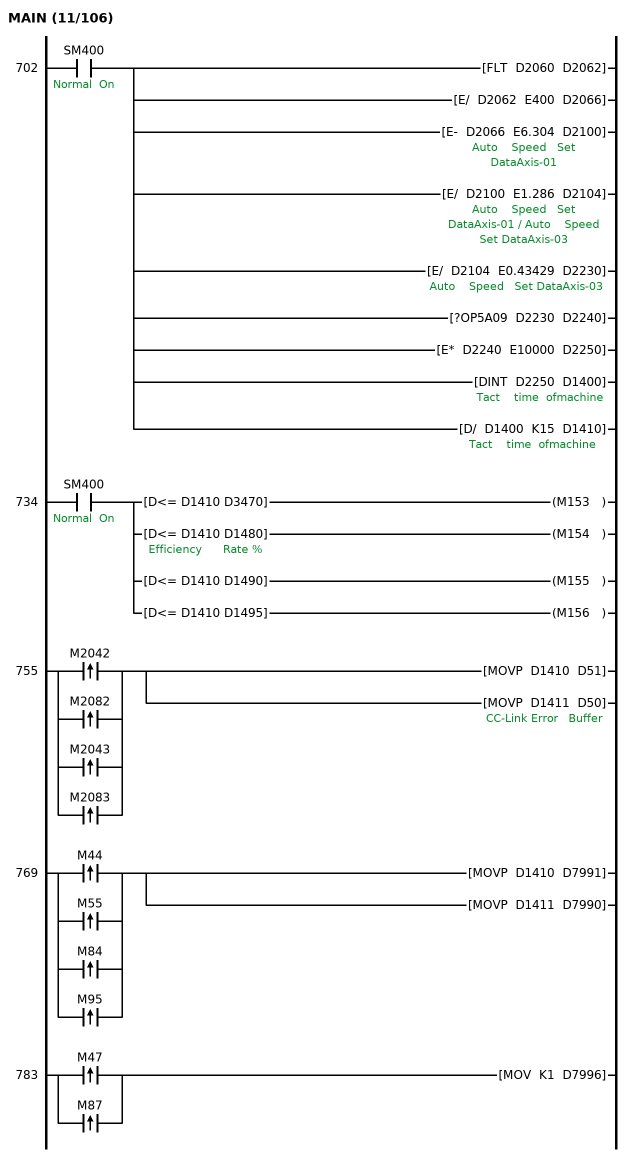
[picture p288: ladder of MAIN, rungs at steps 702 to 783]
702   LD      SM400  ; Normal  On
      FLT     D2060 D2062
      E/      D2062 E400 D2066
      E-      D2066 E6.304 D2100  ; Auto    Speed   Set DataAxis-01
      E/      D2100 E1.286 D2104  ; Auto    Speed   Set DataAxis-03
      E/      D2104 E0.43429 D2230
      ?OP5A09 D2230 D2240
      E*      D2240 E10000 D2250
      DINT    D2250 D1400  ; Tact    time  ofmachine
      D/      D1400 K15 D1410
734   LD      SM400  ; Normal  On
      MPS
      ANDD<=  D1410 D3470
      OUT     M153
      MRD
      ANDD<=  D1410 D1480  ; Efficiency      Rate %
      OUT     M154
      MRD
      ANDD<=  D1410 D1490
      OUT     M155
      MPP
      ANDD<=  D1410 D1495
      OUT     M156
755   LDP     M2042
      ORP     M2082
      ORP     M2043
      ORP     M2083
      MOVP    D1410 D51
      MOVP    D1411 D50  ; CC-Link Error   Buffer
769   LDP     M44
      ORP     M55
      ORP     M84
      ORP     M95
      MOVP    D1410 D7991
      MOVP    D1411 D7990
783   LDP     M47
      ORP     M87
      MOV     K1 D7996
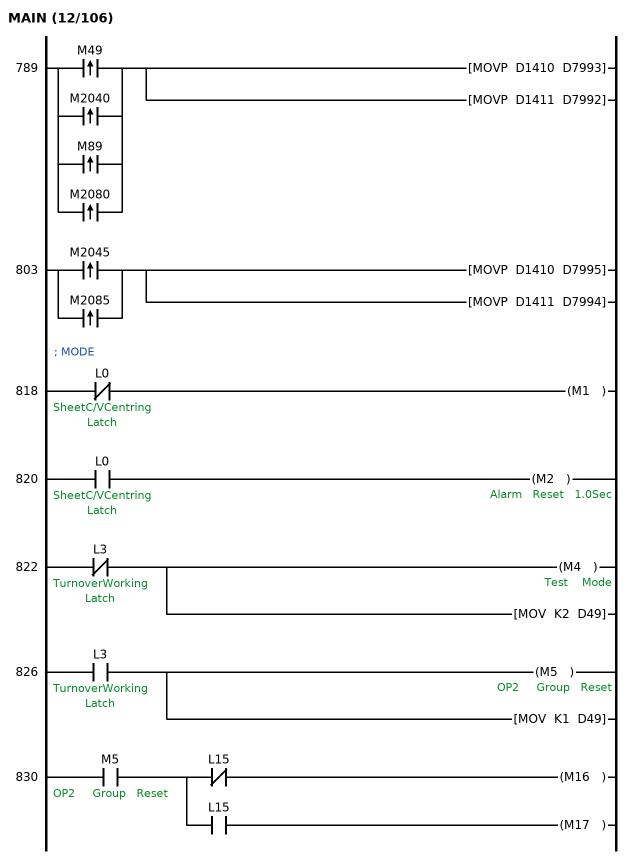
789   LDP     M49
      ORP     M2040
      ORP     M89
      ORP     M2080
      MOVP    D1410 D7993
      MOVP    D1411 D7992
803   LDP     M2045
      ORP     M2085
      MOVP    D1410 D7995
      MOVP    D1411 D7994
; MODE
818   LDI     L0  ; SheetC/VCentringLatch
      OUT     M1
820   LD      L0  ; SheetC/VCentringLatch
      OUT     M2  ; Alarm   Reset   1.0Sec
822   LDI     L3  ; TurnoverWorking Latch
      OUT     M4  ; Test    Mode
      MOV     K2 D49
826   LD      L3  ; TurnoverWorking Latch
      OUT     M5  ; OP2     Group   Reset
      MOV     K1 D49
830   LD      M5  ; OP2     Group   Reset
      MPS
      ANI     L15
      OUT     M16
      MPP
      AND     L15
      OUT     M17
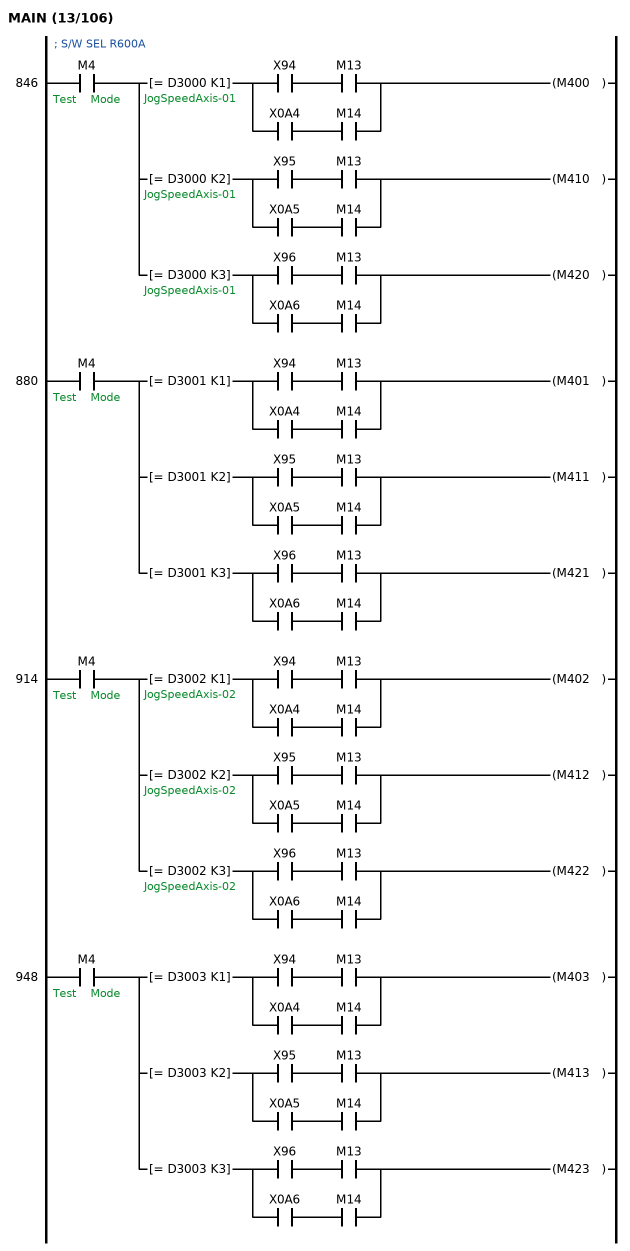
; S/W SEL R600A
846   LD      M4  ; Test    Mode
      MPS
      AND=    D3000 K1  ; JogSpeedAxis-01
      LD      X94
      AND     M13
      LD      X0A4
      AND     M14
      ORB
      ANB
      OUT     M400
      MRD
      AND=    D3000 K2  ; JogSpeedAxis-01
      LD      X95
      AND     M13
      LD      X0A5
      AND     M14
      ORB
      ANB
      OUT     M410
      MPP
      AND=    D3000 K3  ; JogSpeedAxis-01
      LD      X96
      AND     M13
      LD      X0A6
      AND     M14
      ORB
      ANB
      OUT     M420
880   LD      M4  ; Test    Mode
      MPS
      AND=    D3001 K1
      LD      X94
      AND     M13
      LD      X0A4
      AND     M14
      ORB
      ANB
      OUT     M401
      MRD
      AND=    D3001 K2
      LD      X95
      AND     M13
      LD      X0A5
      AND     M14
      ORB
      ANB
      OUT     M411
      MPP
      AND=    D3001 K3
      LD      X96
      AND     M13
      LD      X0A6
      AND     M14
      ORB
      ANB
      OUT     M421
914   LD      M4  ; Test    Mode
      MPS
      AND=    D3002 K1  ; JogSpeedAxis-02
      LD      X94
      AND     M13
      LD      X0A4
      AND     M14
      ORB
      ANB
      OUT     M402
      MRD
      AND=    D3002 K2  ; JogSpeedAxis-02
      LD      X95
      AND     M13
      LD      X0A5
      AND     M14
      ORB
      ANB
      OUT     M412
      MPP
      AND=    D3002 K3  ; JogSpeedAxis-02
      LD      X96
      AND     M13
      LD      X0A6
      AND     M14
      ORB
      ANB
      OUT     M422
948   LD      M4  ; Test    Mode
      MPS
      AND=    D3003 K1
      LD      X94
      AND     M13
      LD      X0A4
      AND     M14
      ORB
      ANB
      OUT     M403
      MRD
      AND=    D3003 K2
      LD      X95
      AND     M13
      LD      X0A5
      AND     M14
      ORB
      ANB
      OUT     M413
      MPP
      AND=    D3003 K3
      LD      X96
      AND     M13
      LD      X0A6
      AND     M14
      ORB
      ANB
      OUT     M423
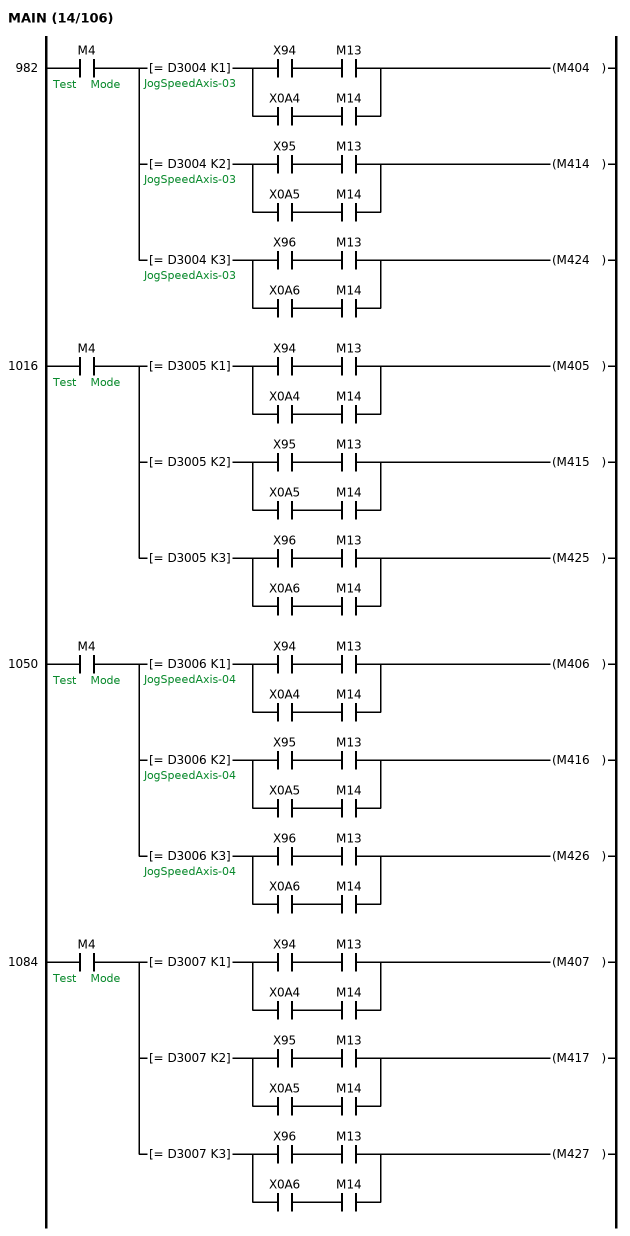
982   LD      M4  ; Test    Mode
      MPS
      AND=    D3004 K1  ; JogSpeedAxis-03
      LD      X94
      AND     M13
      LD      X0A4
      AND     M14
      ORB
      ANB
      OUT     M404
      MRD
      AND=    D3004 K2  ; JogSpeedAxis-03
      LD      X95
      AND     M13
      LD      X0A5
      AND     M14
      ORB
      ANB
      OUT     M414
      MPP
      AND=    D3004 K3  ; JogSpeedAxis-03
      LD      X96
      AND     M13
      LD      X0A6
      AND     M14
      ORB
      ANB
      OUT     M424
1016  LD      M4  ; Test    Mode
      MPS
      AND=    D3005 K1
      LD      X94
      AND     M13
      LD      X0A4
      AND     M14
      ORB
      ANB
      OUT     M405
      MRD
      AND=    D3005 K2
      LD      X95
      AND     M13
      LD      X0A5
      AND     M14
      ORB
      ANB
      OUT     M415
      MPP
      AND=    D3005 K3
      LD      X96
      AND     M13
      LD      X0A6
      AND     M14
      ORB
      ANB
      OUT     M425
1050  LD      M4  ; Test    Mode
      MPS
      AND=    D3006 K1  ; JogSpeedAxis-04
      LD      X94
      AND     M13
      LD      X0A4
      AND     M14
      ORB
      ANB
      OUT     M406
      MRD
      AND=    D3006 K2  ; JogSpeedAxis-04
      LD      X95
      AND     M13
      LD      X0A5
      AND     M14
      ORB
      ANB
      OUT     M416
      MPP
      AND=    D3006 K3  ; JogSpeedAxis-04
      LD      X96
      AND     M13
      LD      X0A6
      AND     M14
      ORB
      ANB
      OUT     M426
1084  LD      M4  ; Test    Mode
      MPS
      AND=    D3007 K1
      LD      X94
      AND     M13
      LD      X0A4
      AND     M14
      ORB
      ANB
      OUT     M407
      MRD
      AND=    D3007 K2
      LD      X95
      AND     M13
      LD      X0A5
      AND     M14
      ORB
      ANB
      OUT     M417
      MPP
      AND=    D3007 K3
      LD      X96
      AND     M13
      LD      X0A6
      AND     M14
      ORB
      ANB
      OUT     M427
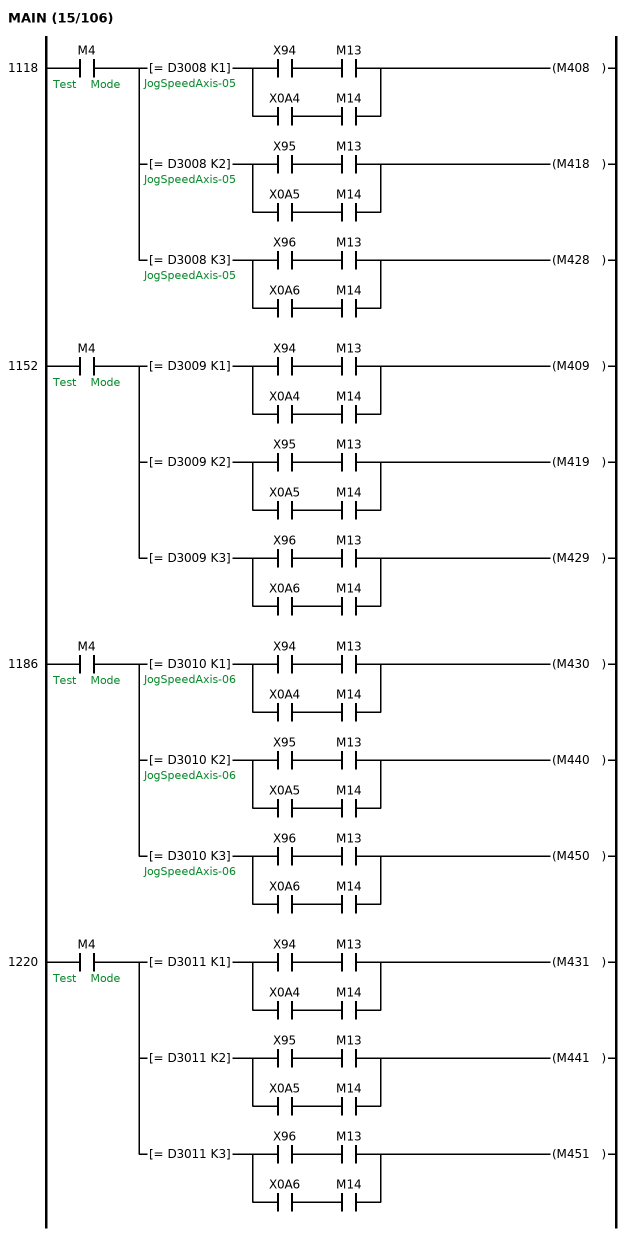
1118  LD      M4  ; Test    Mode
      MPS
      AND=    D3008 K1  ; JogSpeedAxis-05
      LD      X94
      AND     M13
      LD      X0A4
      AND     M14
      ORB
      ANB
      OUT     M408
      MRD
      AND=    D3008 K2  ; JogSpeedAxis-05
      LD      X95
      AND     M13
      LD      X0A5
      AND     M14
      ORB
      ANB
      OUT     M418
      MPP
      AND=    D3008 K3  ; JogSpeedAxis-05
      LD      X96
      AND     M13
      LD      X0A6
      AND     M14
      ORB
      ANB
      OUT     M428
1152  LD      M4  ; Test    Mode
      MPS
      AND=    D3009 K1
      LD      X94
      AND     M13
      LD      X0A4
      AND     M14
      ORB
      ANB
      OUT     M409
      MRD
      AND=    D3009 K2
      LD      X95
      AND     M13
      LD      X0A5
      AND     M14
      ORB
      ANB
      OUT     M419
      MPP
      AND=    D3009 K3
      LD      X96
      AND     M13
      LD      X0A6
      AND     M14
      ORB
      ANB
      OUT     M429
1186  LD      M4  ; Test    Mode
      MPS
      AND=    D3010 K1  ; JogSpeedAxis-06
      LD      X94
      AND     M13
      LD      X0A4
      AND     M14
      ORB
      ANB
      OUT     M430
      MRD
      AND=    D3010 K2  ; JogSpeedAxis-06
      LD      X95
      AND     M13
      LD      X0A5
      AND     M14
      ORB
      ANB
      OUT     M440
      MPP
      AND=    D3010 K3  ; JogSpeedAxis-06
      LD      X96
      AND     M13
      LD      X0A6
      AND     M14
      ORB
      ANB
      OUT     M450
1220  LD      M4  ; Test    Mode
      MPS
      AND=    D3011 K1
      LD      X94
      AND     M13
      LD      X0A4
      AND     M14
      ORB
      ANB
      OUT     M431
      MRD
      AND=    D3011 K2
      LD      X95
      AND     M13
      LD      X0A5
      AND     M14
      ORB
      ANB
      OUT     M441
      MPP
      AND=    D3011 K3
      LD      X96
      AND     M13
      LD      X0A6
      AND     M14
      ORB
      ANB
      OUT     M451
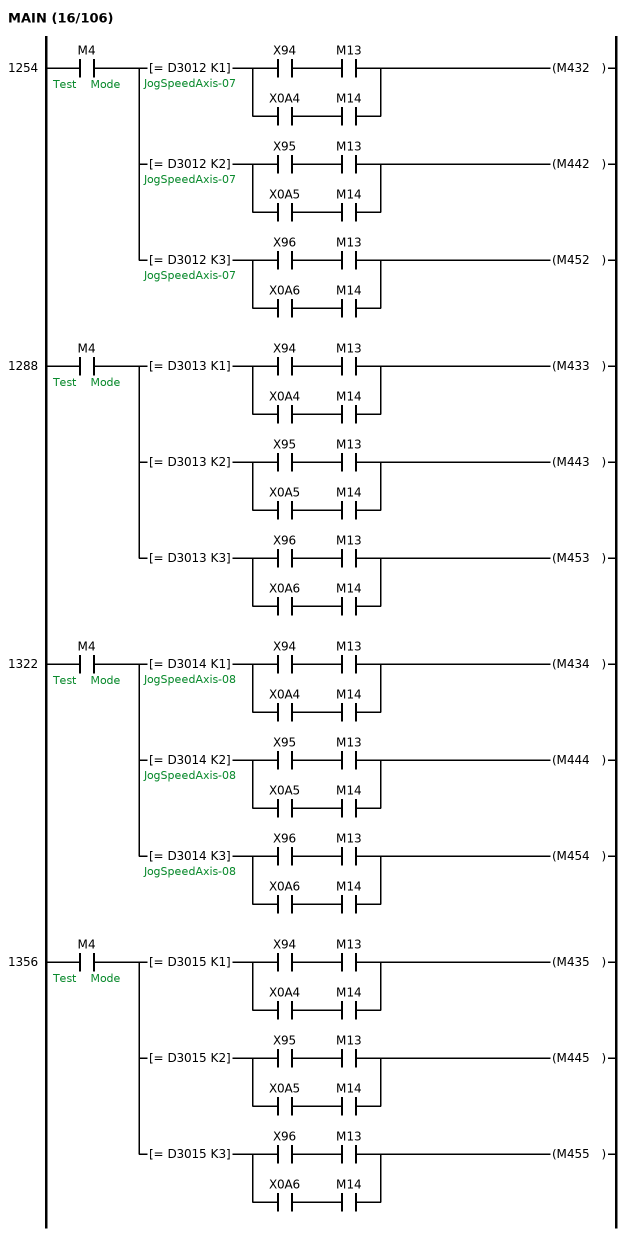
1254  LD      M4  ; Test    Mode
      MPS
      AND=    D3012 K1  ; JogSpeedAxis-07
      LD      X94
      AND     M13
      LD      X0A4
      AND     M14
      ORB
      ANB
      OUT     M432
      MRD
      AND=    D3012 K2  ; JogSpeedAxis-07
      LD      X95
      AND     M13
      LD      X0A5
      AND     M14
      ORB
      ANB
      OUT     M442
      MPP
      AND=    D3012 K3  ; JogSpeedAxis-07
      LD      X96
      AND     M13
      LD      X0A6
      AND     M14
      ORB
      ANB
      OUT     M452
1288  LD      M4  ; Test    Mode
      MPS
      AND=    D3013 K1
      LD      X94
      AND     M13
      LD      X0A4
      AND     M14
      ORB
      ANB
      OUT     M433
      MRD
      AND=    D3013 K2
      LD      X95
      AND     M13
      LD      X0A5
      AND     M14
      ORB
      ANB
      OUT     M443
      MPP
      AND=    D3013 K3
      LD      X96
      AND     M13
      LD      X0A6
      AND     M14
      ORB
      ANB
      OUT     M453
1322  LD      M4  ; Test    Mode
      MPS
      AND=    D3014 K1  ; JogSpeedAxis-08
      LD      X94
      AND     M13
      LD      X0A4
      AND     M14
      ORB
      ANB
      OUT     M434
      MRD
      AND=    D3014 K2  ; JogSpeedAxis-08
      LD      X95
      AND     M13
      LD      X0A5
      AND     M14
      ORB
      ANB
      OUT     M444
      MPP
      AND=    D3014 K3  ; JogSpeedAxis-08
      LD      X96
      AND     M13
      LD      X0A6
      AND     M14
      ORB
      ANB
      OUT     M454
1356  LD      M4  ; Test    Mode
      MPS
      AND=    D3015 K1
      LD      X94
      AND     M13
      LD      X0A4
      AND     M14
      ORB
      ANB
      OUT     M435
      MRD
      AND=    D3015 K2
      LD      X95
      AND     M13
      LD      X0A5
      AND     M14
      ORB
      ANB
      OUT     M445
      MPP
      AND=    D3015 K3
      LD      X96
      AND     M13
      LD      X0A6
      AND     M14
      ORB
      ANB
      OUT     M455
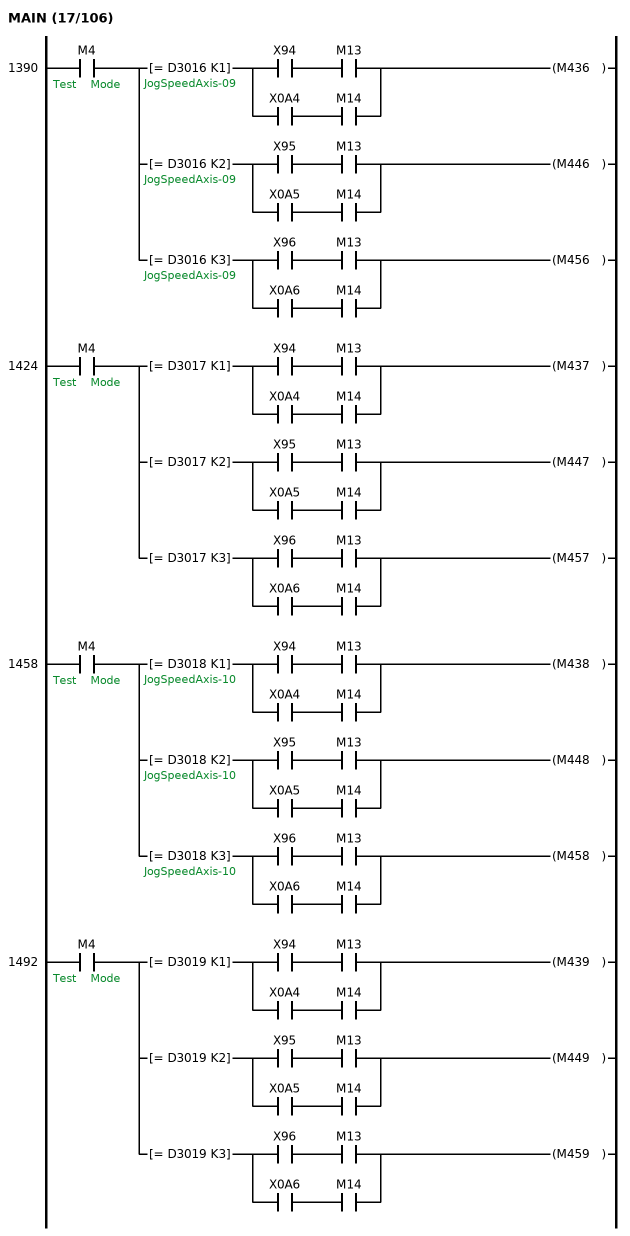
1390  LD      M4  ; Test    Mode
      MPS
      AND=    D3016 K1  ; JogSpeedAxis-09
      LD      X94
      AND     M13
      LD      X0A4
      AND     M14
      ORB
      ANB
      OUT     M436
      MRD
      AND=    D3016 K2  ; JogSpeedAxis-09
      LD      X95
      AND     M13
      LD      X0A5
      AND     M14
      ORB
      ANB
      OUT     M446
      MPP
      AND=    D3016 K3  ; JogSpeedAxis-09
      LD      X96
      AND     M13
      LD      X0A6
      AND     M14
      ORB
      ANB
      OUT     M456
1424  LD      M4  ; Test    Mode
      MPS
      AND=    D3017 K1
      LD      X94
      AND     M13
      LD      X0A4
      AND     M14
      ORB
      ANB
      OUT     M437
      MRD
      AND=    D3017 K2
      LD      X95
      AND     M13
      LD      X0A5
      AND     M14
      ORB
      ANB
      OUT     M447
      MPP
      AND=    D3017 K3
      LD      X96
      AND     M13
      LD      X0A6
      AND     M14
      ORB
      ANB
      OUT     M457
1458  LD      M4  ; Test    Mode
      MPS
      AND=    D3018 K1  ; JogSpeedAxis-10
      LD      X94
      AND     M13
      LD      X0A4
      AND     M14
      ORB
      ANB
      OUT     M438
      MRD
      AND=    D3018 K2  ; JogSpeedAxis-10
      LD      X95
      AND     M13
      LD      X0A5
      AND     M14
      ORB
      ANB
      OUT     M448
      MPP
      AND=    D3018 K3  ; JogSpeedAxis-10
      LD      X96
      AND     M13
      LD      X0A6
      AND     M14
      ORB
      ANB
      OUT     M458
1492  LD      M4  ; Test    Mode
      MPS
      AND=    D3019 K1
      LD      X94
      AND     M13
      LD      X0A4
      AND     M14
      ORB
      ANB
      OUT     M439
      MRD
      AND=    D3019 K2
      LD      X95
      AND     M13
      LD      X0A5
      AND     M14
      ORB
      ANB
      OUT     M449
      MPP
      AND=    D3019 K3
      LD      X96
      AND     M13
      LD      X0A6
      AND     M14
      ORB
      ANB
      OUT     M459
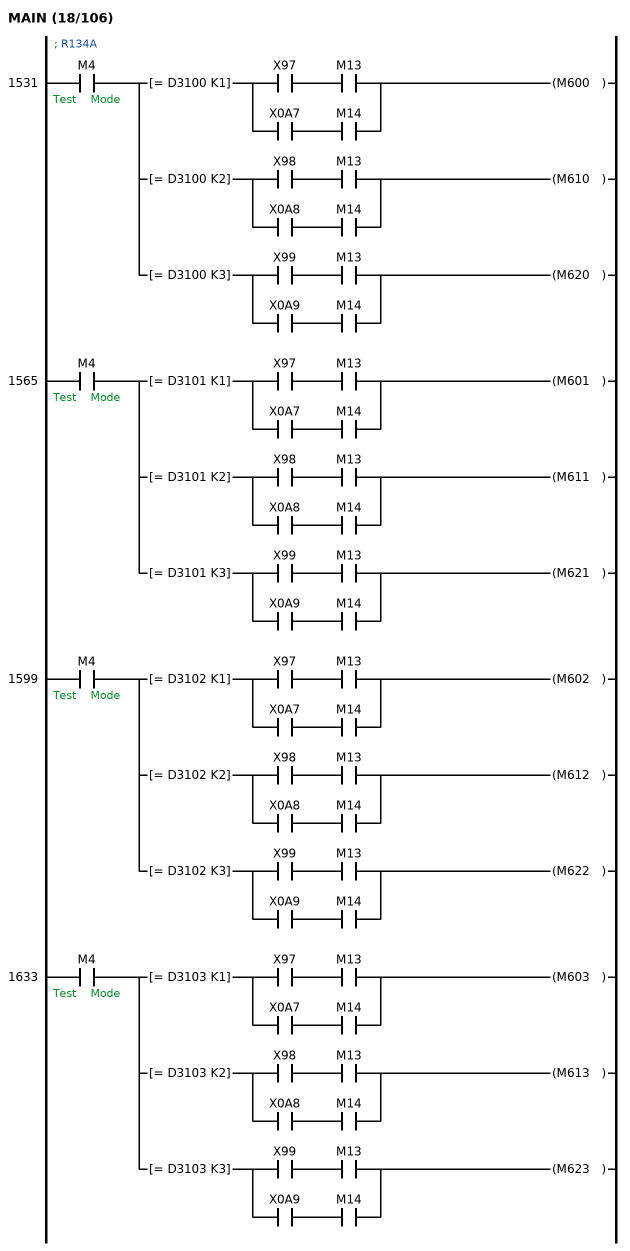
; R134A
1531  LD      M4  ; Test    Mode
      MPS
      AND=    D3100 K1
      LD      X97
      AND     M13
      LD      X0A7
      AND     M14
      ORB
      ANB
      OUT     M600
      MRD
      AND=    D3100 K2
      LD      X98
      AND     M13
      LD      X0A8
      AND     M14
      ORB
      ANB
      OUT     M610
      MPP
      AND=    D3100 K3
      LD      X99
      AND     M13
      LD      X0A9
      AND     M14
      ORB
      ANB
      OUT     M620
1565  LD      M4  ; Test    Mode
      MPS
      AND=    D3101 K1
      LD      X97
      AND     M13
      LD      X0A7
      AND     M14
      ORB
      ANB
      OUT     M601
      MRD
      AND=    D3101 K2
      LD      X98
      AND     M13
      LD      X0A8
      AND     M14
      ORB
      ANB
      OUT     M611
      MPP
      AND=    D3101 K3
      LD      X99
      AND     M13
      LD      X0A9
      AND     M14
      ORB
      ANB
      OUT     M621
1599  LD      M4  ; Test    Mode
      MPS
      AND=    D3102 K1
      LD      X97
      AND     M13
      LD      X0A7
      AND     M14
      ORB
      ANB
      OUT     M602
      MRD
      AND=    D3102 K2
      LD      X98
      AND     M13
      LD      X0A8
      AND     M14
      ORB
      ANB
      OUT     M612
      MPP
      AND=    D3102 K3
      LD      X99
      AND     M13
      LD      X0A9
      AND     M14
      ORB
      ANB
      OUT     M622
1633  LD      M4  ; Test    Mode
      MPS
      AND=    D3103 K1
      LD      X97
      AND     M13
      LD      X0A7
      AND     M14
      ORB
      ANB
      OUT     M603
      MRD
      AND=    D3103 K2
      LD      X98
      AND     M13
      LD      X0A8
      AND     M14
      ORB
      ANB
      OUT     M613
      MPP
      AND=    D3103 K3
      LD      X99
      AND     M13
      LD      X0A9
      AND     M14
      ORB
      ANB
      OUT     M623
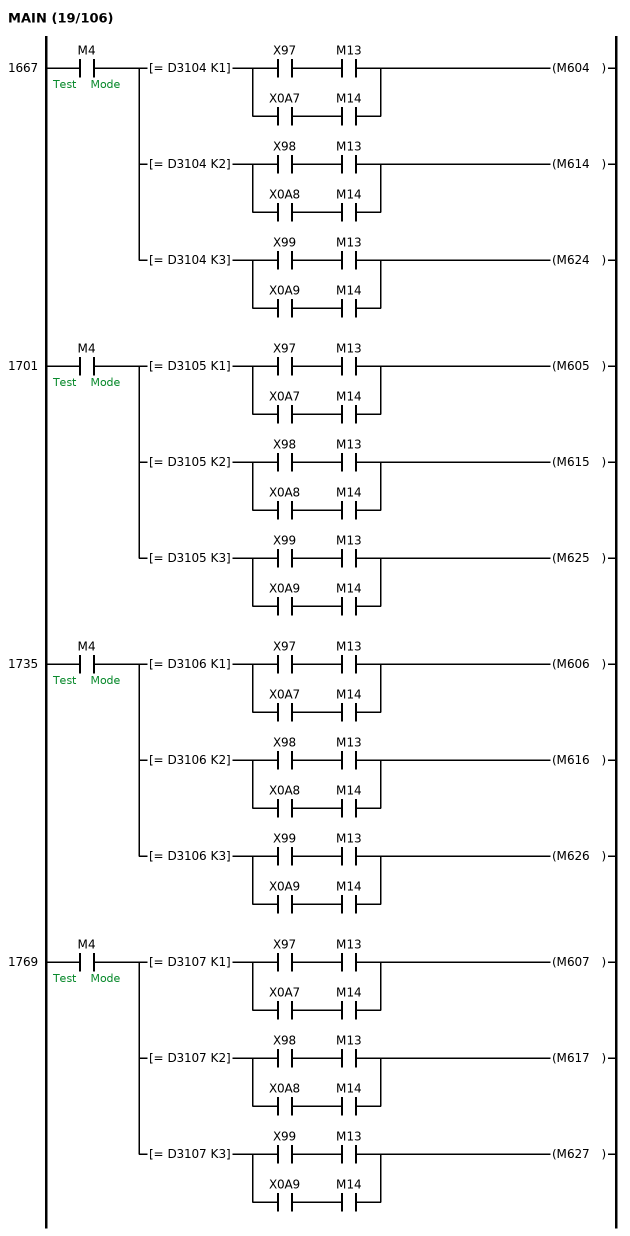
1667  LD      M4  ; Test    Mode
      MPS
      AND=    D3104 K1
      LD      X97
      AND     M13
      LD      X0A7
      AND     M14
      ORB
      ANB
      OUT     M604
      MRD
      AND=    D3104 K2
      LD      X98
      AND     M13
      LD      X0A8
      AND     M14
      ORB
      ANB
      OUT     M614
      MPP
      AND=    D3104 K3
      LD      X99
      AND     M13
      LD      X0A9
      AND     M14
      ORB
      ANB
      OUT     M624
1701  LD      M4  ; Test    Mode
      MPS
      AND=    D3105 K1
      LD      X97
      AND     M13
      LD      X0A7
      AND     M14
      ORB
      ANB
      OUT     M605
      MRD
      AND=    D3105 K2
      LD      X98
      AND     M13
      LD      X0A8
      AND     M14
      ORB
      ANB
      OUT     M615
      MPP
      AND=    D3105 K3
      LD      X99
      AND     M13
      LD      X0A9
      AND     M14
      ORB
      ANB
      OUT     M625
1735  LD      M4  ; Test    Mode
      MPS
      AND=    D3106 K1
      LD      X97
      AND     M13
      LD      X0A7
      AND     M14
      ORB
      ANB
      OUT     M606
      MRD
      AND=    D3106 K2
      LD      X98
      AND     M13
      LD      X0A8
      AND     M14
      ORB
      ANB
      OUT     M616
      MPP
      AND=    D3106 K3
      LD      X99
      AND     M13
      LD      X0A9
      AND     M14
      ORB
      ANB
      OUT     M626
1769  LD      M4  ; Test    Mode
      MPS
      AND=    D3107 K1
      LD      X97
      AND     M13
      LD      X0A7
      AND     M14
      ORB
      ANB
      OUT     M607
      MRD
      AND=    D3107 K2
      LD      X98
      AND     M13
      LD      X0A8
      AND     M14
      ORB
      ANB
      OUT     M617
      MPP
      AND=    D3107 K3
      LD      X99
      AND     M13
      LD      X0A9
      AND     M14
      ORB
      ANB
      OUT     M627
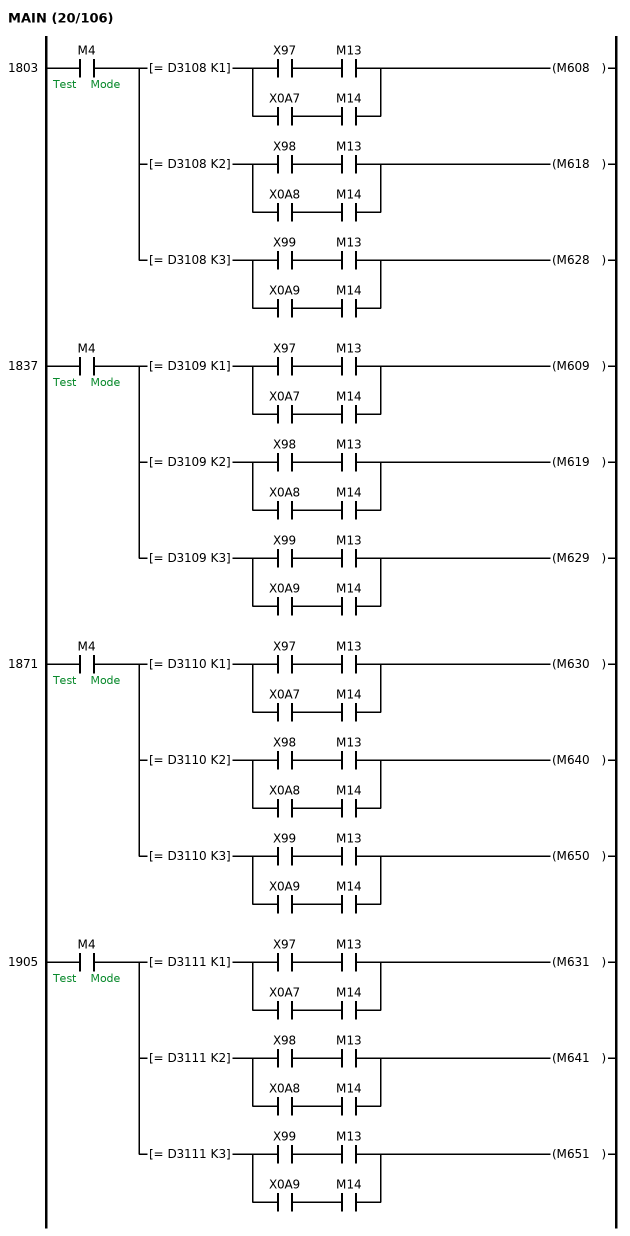
1803  LD      M4  ; Test    Mode
      MPS
      AND=    D3108 K1
      LD      X97
      AND     M13
      LD      X0A7
      AND     M14
      ORB
      ANB
      OUT     M608
      MRD
      AND=    D3108 K2
      LD      X98
      AND     M13
      LD      X0A8
      AND     M14
      ORB
      ANB
      OUT     M618
      MPP
      AND=    D3108 K3
      LD      X99
      AND     M13
      LD      X0A9
      AND     M14
      ORB
      ANB
      OUT     M628
1837  LD      M4  ; Test    Mode
      MPS
      AND=    D3109 K1
      LD      X97
      AND     M13
      LD      X0A7
      AND     M14
      ORB
      ANB
      OUT     M609
      MRD
      AND=    D3109 K2
      LD      X98
      AND     M13
      LD      X0A8
      AND     M14
      ORB
      ANB
      OUT     M619
      MPP
      AND=    D3109 K3
      LD      X99
      AND     M13
      LD      X0A9
      AND     M14
      ORB
      ANB
      OUT     M629
1871  LD      M4  ; Test    Mode
      MPS
      AND=    D3110 K1
      LD      X97
      AND     M13
      LD      X0A7
      AND     M14
      ORB
      ANB
      OUT     M630
      MRD
      AND=    D3110 K2
      LD      X98
      AND     M13
      LD      X0A8
      AND     M14
      ORB
      ANB
      OUT     M640
      MPP
      AND=    D3110 K3
      LD      X99
      AND     M13
      LD      X0A9
      AND     M14
      ORB
      ANB
      OUT     M650
1905  LD      M4  ; Test    Mode
      MPS
      AND=    D3111 K1
      LD      X97
      AND     M13
      LD      X0A7
      AND     M14
      ORB
      ANB
      OUT     M631
      MRD
      AND=    D3111 K2
      LD      X98
      AND     M13
      LD      X0A8
      AND     M14
      ORB
      ANB
      OUT     M641
      MPP
      AND=    D3111 K3
      LD      X99
      AND     M13
      LD      X0A9
      AND     M14
      ORB
      ANB
      OUT     M651
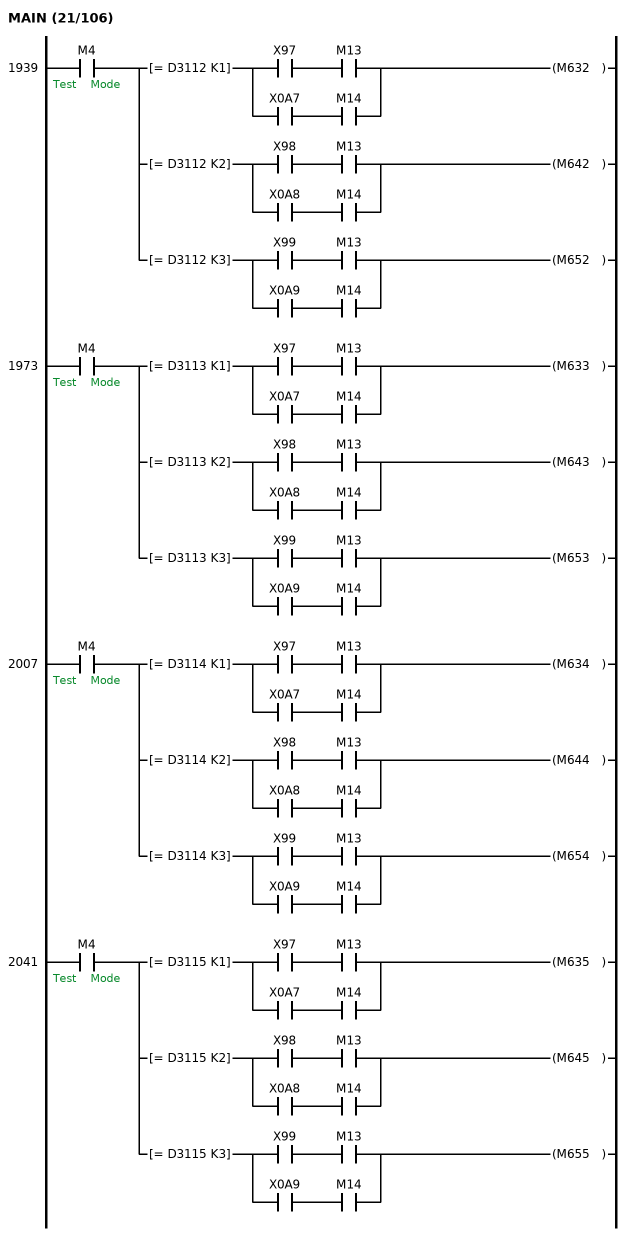
1939  LD      M4  ; Test    Mode
      MPS
      AND=    D3112 K1
      LD      X97
      AND     M13
      LD      X0A7
      AND     M14
      ORB
      ANB
      OUT     M632
      MRD
      AND=    D3112 K2
      LD      X98
      AND     M13
      LD      X0A8
      AND     M14
      ORB
      ANB
      OUT     M642
      MPP
      AND=    D3112 K3
      LD      X99
      AND     M13
      LD      X0A9
      AND     M14
      ORB
      ANB
      OUT     M652
1973  LD      M4  ; Test    Mode
      MPS
      AND=    D3113 K1
      LD      X97
      AND     M13
      LD      X0A7
      AND     M14
      ORB
      ANB
      OUT     M633
      MRD
      AND=    D3113 K2
      LD      X98
      AND     M13
      LD      X0A8
      AND     M14
      ORB
      ANB
      OUT     M643
      MPP
      AND=    D3113 K3
      LD      X99
      AND     M13
      LD      X0A9
      AND     M14
      ORB
      ANB
      OUT     M653
2007  LD      M4  ; Test    Mode
      MPS
      AND=    D3114 K1
      LD      X97
      AND     M13
      LD      X0A7
      AND     M14
      ORB
      ANB
      OUT     M634
      MRD
      AND=    D3114 K2
      LD      X98
      AND     M13
      LD      X0A8
      AND     M14
      ORB
      ANB
      OUT     M644
      MPP
      AND=    D3114 K3
      LD      X99
      AND     M13
      LD      X0A9
      AND     M14
      ORB
      ANB
      OUT     M654
2041  LD      M4  ; Test    Mode
      MPS
      AND=    D3115 K1
      LD      X97
      AND     M13
      LD      X0A7
      AND     M14
      ORB
      ANB
      OUT     M635
      MRD
      AND=    D3115 K2
      LD      X98
      AND     M13
      LD      X0A8
      AND     M14
      ORB
      ANB
      OUT     M645
      MPP
      AND=    D3115 K3
      LD      X99
      AND     M13
      LD      X0A9
      AND     M14
      ORB
      ANB
      OUT     M655
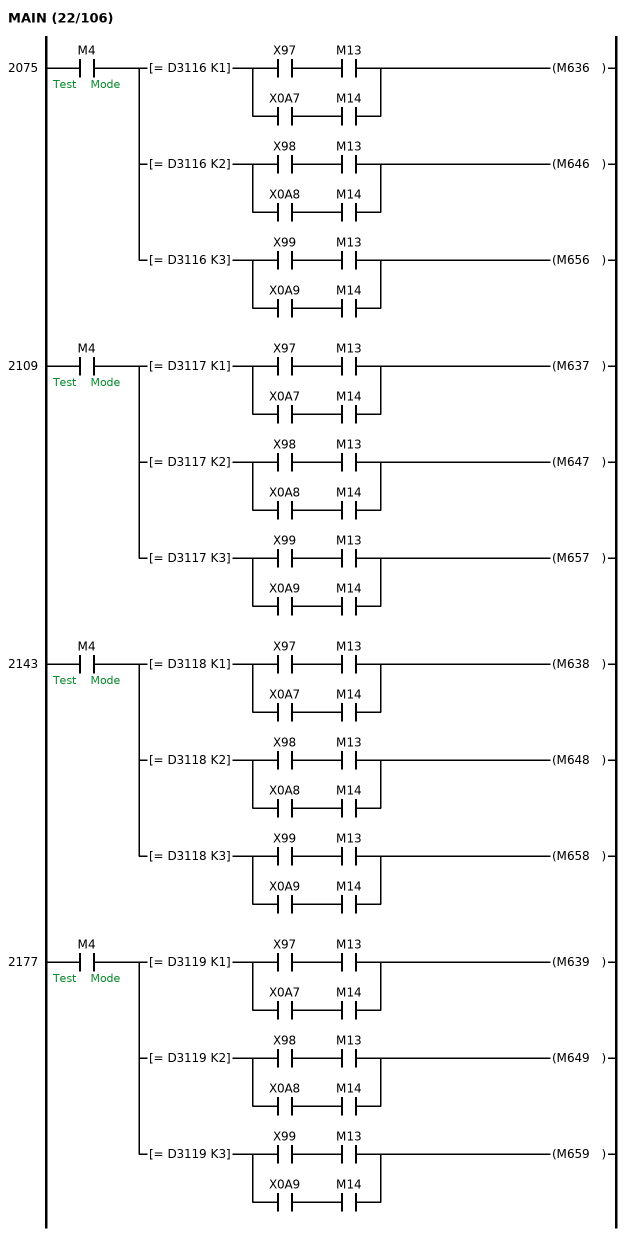
2075  LD      M4  ; Test    Mode
      MPS
      AND=    D3116 K1
      LD      X97
      AND     M13
      LD      X0A7
      AND     M14
      ORB
      ANB
      OUT     M636
      MRD
      AND=    D3116 K2
      LD      X98
      AND     M13
      LD      X0A8
      AND     M14
      ORB
      ANB
      OUT     M646
      MPP
      AND=    D3116 K3
      LD      X99
      AND     M13
      LD      X0A9
      AND     M14
      ORB
      ANB
      OUT     M656
2109  LD      M4  ; Test    Mode
      MPS
      AND=    D3117 K1
      LD      X97
      AND     M13
      LD      X0A7
      AND     M14
      ORB
      ANB
      OUT     M637
      MRD
      AND=    D3117 K2
      LD      X98
      AND     M13
      LD      X0A8
      AND     M14
      ORB
      ANB
      OUT     M647
      MPP
      AND=    D3117 K3
      LD      X99
      AND     M13
      LD      X0A9
      AND     M14
      ORB
      ANB
      OUT     M657
2143  LD      M4  ; Test    Mode
      MPS
      AND=    D3118 K1
      LD      X97
      AND     M13
      LD      X0A7
      AND     M14
      ORB
      ANB
      OUT     M638
      MRD
      AND=    D3118 K2
      LD      X98
      AND     M13
      LD      X0A8
      AND     M14
      ORB
      ANB
      OUT     M648
      MPP
      AND=    D3118 K3
      LD      X99
      AND     M13
      LD      X0A9
      AND     M14
      ORB
      ANB
      OUT     M658
2177  LD      M4  ; Test    Mode
      MPS
      AND=    D3119 K1
      LD      X97
      AND     M13
      LD      X0A7
      AND     M14
      ORB
      ANB
      OUT     M639
      MRD
      AND=    D3119 K2
      LD      X98
      AND     M13
      LD      X0A8
      AND     M14
      ORB
      ANB
      OUT     M649
      MPP
      AND=    D3119 K3
      LD      X99
      AND     M13
      LD      X0A9
      AND     M14
      ORB
      ANB
      OUT     M659
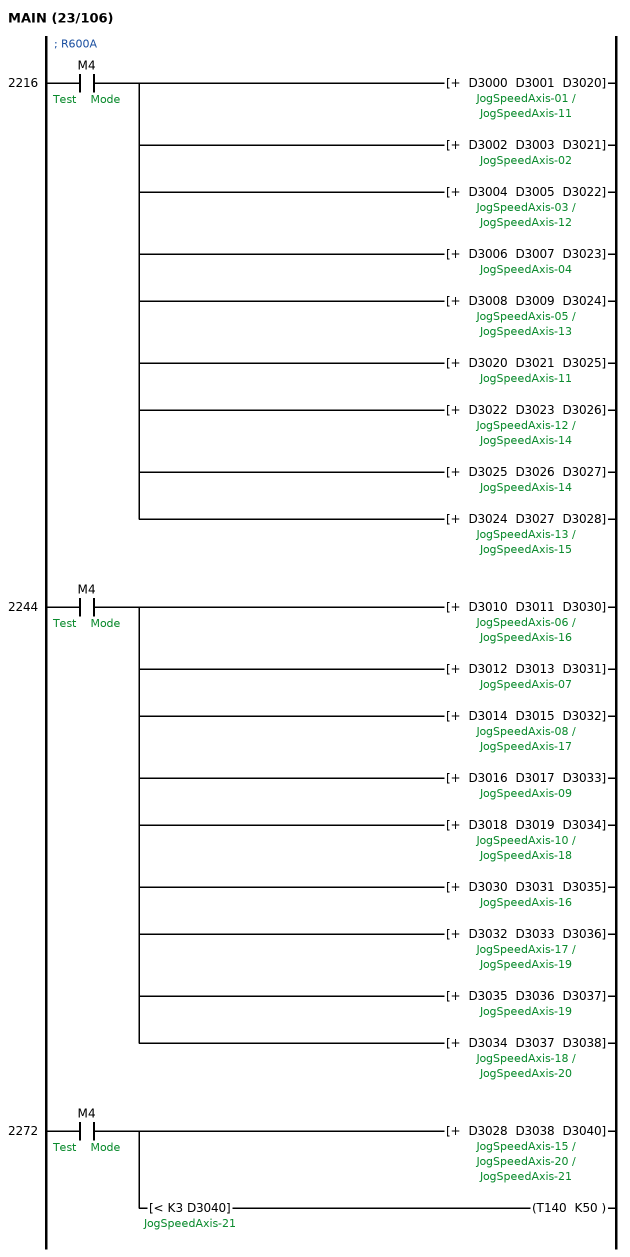
; R600A
2216  LD      M4  ; Test    Mode
      +       D3000 D3001 D3020  ; JogSpeedAxis-11
      +       D3002 D3003 D3021
      +       D3004 D3005 D3022  ; JogSpeedAxis-12
      +       D3006 D3007 D3023
      +       D3008 D3009 D3024  ; JogSpeedAxis-13
      +       D3020 D3021 D3025
      +       D3022 D3023 D3026  ; JogSpeedAxis-14
      +       D3025 D3026 D3027
      +       D3024 D3027 D3028  ; JogSpeedAxis-15
2244  LD      M4  ; Test    Mode
      +       D3010 D3011 D3030  ; JogSpeedAxis-16
      +       D3012 D3013 D3031
      +       D3014 D3015 D3032  ; JogSpeedAxis-17
      +       D3016 D3017 D3033
      +       D3018 D3019 D3034  ; JogSpeedAxis-18
      +       D3030 D3031 D3035
      +       D3032 D3033 D3036  ; JogSpeedAxis-19
      +       D3035 D3036 D3037
      +       D3034 D3037 D3038  ; JogSpeedAxis-20
2272  LD      M4  ; Test    Mode
      +       D3028 D3038 D3040  ; JogSpeedAxis-21
      AND<    K3 D3040  ; JogSpeedAxis-21
      OUT     T140 K50
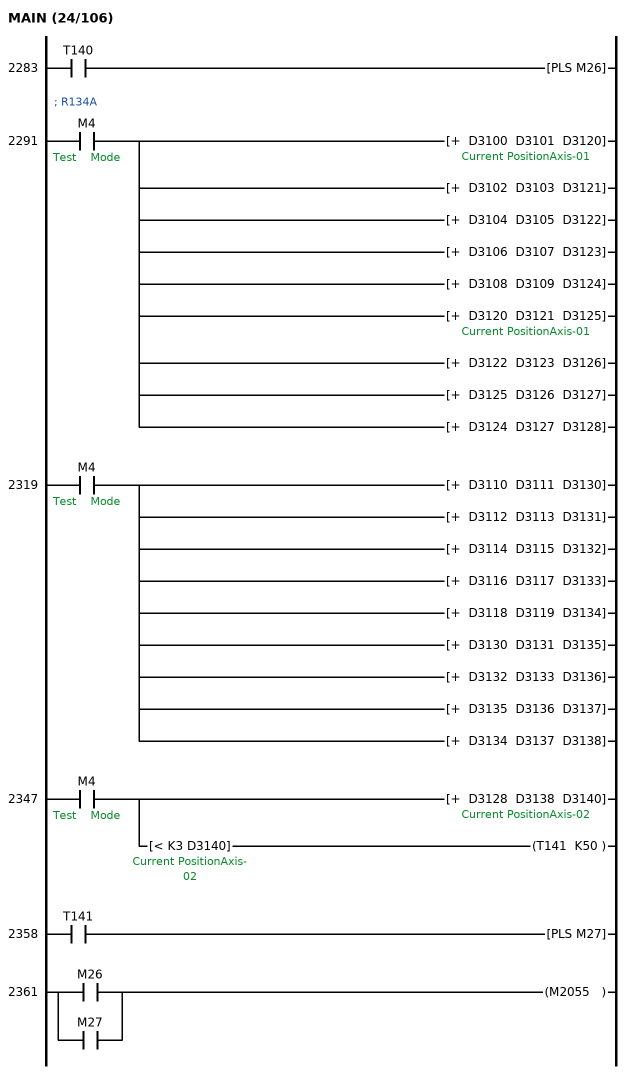
2283  LD      T140
      PLS     M26
; R134A
2291  LD      M4  ; Test    Mode
      +       D3100 D3101 D3120  ; Current PositionAxis-01
      +       D3102 D3103 D3121
      +       D3104 D3105 D3122
      +       D3106 D3107 D3123
      +       D3108 D3109 D3124
      +       D3120 D3121 D3125
      +       D3122 D3123 D3126
      +       D3125 D3126 D3127
      +       D3124 D3127 D3128
2319  LD      M4  ; Test    Mode
      +       D3110 D3111 D3130
      +       D3112 D3113 D3131
      +       D3114 D3115 D3132
      +       D3116 D3117 D3133
      +       D3118 D3119 D3134
      +       D3130 D3131 D3135
      +       D3132 D3133 D3136
      +       D3135 D3136 D3137
      +       D3134 D3137 D3138
2347  LD      M4  ; Test    Mode
      +       D3128 D3138 D3140  ; Current PositionAxis-02
      AND<    K3 D3140  ; Current PositionAxis-02
      OUT     T141 K50
2358  LD      T141
      PLS     M27
2361  LD      M26
      OR      M27
      OUT     M2055
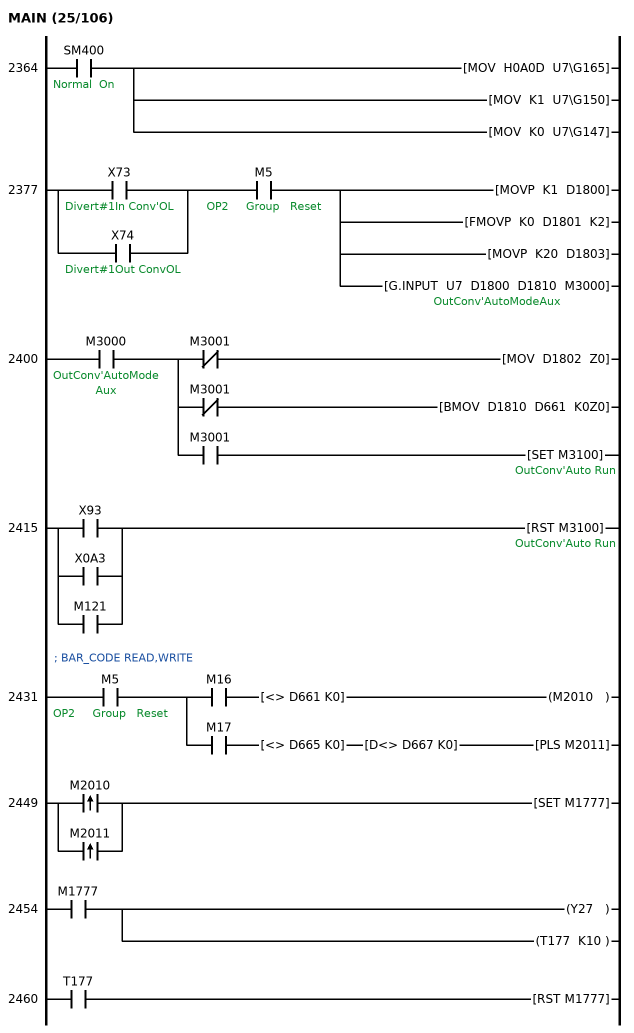
2364  LD      SM400  ; Normal  On
      MOV     H0A0D U7\G165
      MOV     K1 U7\G150
      MOV     K0 U7\G147
2377  LD      X73  ; Divert#1In Conv'OL
      OR      X74  ; Divert#1Out ConvOL
      AND     M5  ; OP2     Group   Reset
      MOVP    K1 D1800
      FMOVP   K0 D1801 K2
      MOVP    K20 D1803
      G.INPUT U7 D1800 D1810 M3000  ; OutConv'AutoModeAux
2400  LD      M3000  ; OutConv'AutoModeAux
      MPS
      ANI     M3001
      MOV     D1802 Z0
      MRD
      ANI     M3001
      BMOV    D1810 D661 K0Z0
      MPP
      AND     M3001
      SET     M3100  ; OutConv'Auto Run
2415  LD      X93
      OR      X0A3
      OR      M121
      RST     M3100  ; OutConv'Auto Run
; BAR_CODE READ,WRITE
2431  LD      M5  ; OP2     Group   Reset
      MPS
      AND     M16
      AND<>   D661 K0
      OUT     M2010
      MPP
      AND     M17
      AND<>   D665 K0
      ANDD<>  D667 K0
      PLS     M2011
2449  LDP     M2010
      ORP     M2011
      SET     M1777
2454  LD      M1777
      OUT     Y27
      OUT     T177 K10
2460  LD      T177
      RST     M1777
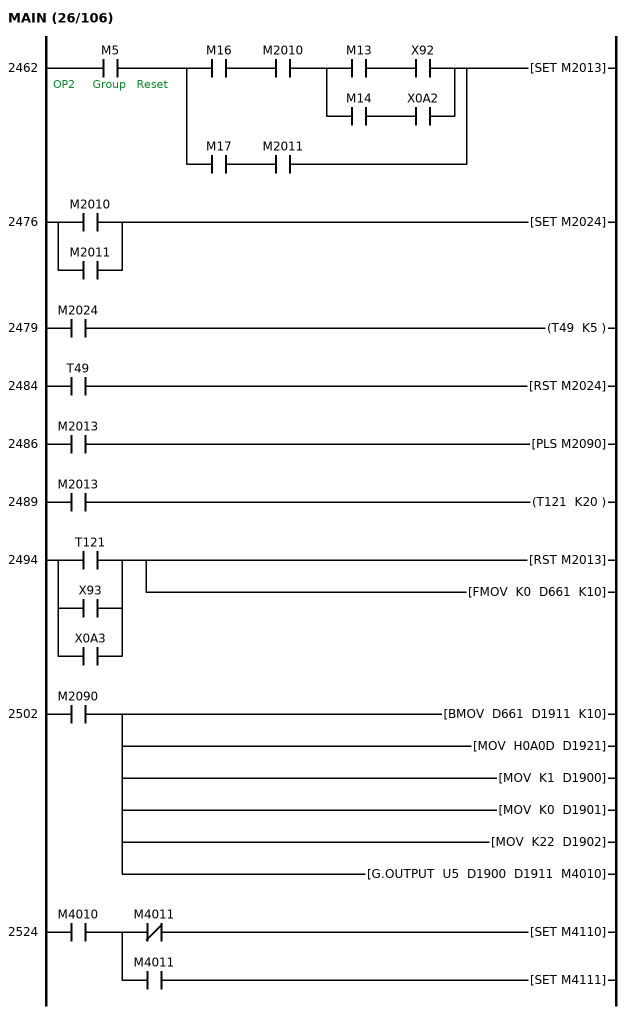
2462  LD      M5  ; OP2     Group   Reset
      LD      M16
      AND     M2010
      LD      M13
      AND     X92
      LD      M14
      AND     X0A2
      ORB
      ANB
      LD      M17
      AND     M2011
      ORB
      ANB
      SET     M2013
2476  LD      M2010
      OR      M2011
      SET     M2024
2479  LD      M2024
      OUT     T49 K5
2484  LD      T49
      RST     M2024
2486  LD      M2013
      PLS     M2090
2489  LD      M2013
      OUT     T121 K20
2494  LD      T121
      OR      X93
      OR      X0A3
      RST     M2013
      FMOV    K0 D661 K10
2502  LD      M2090
      BMOV    D661 D1911 K10
      MOV     H0A0D D1921
      MOV     K1 D1900
      MOV     K0 D1901
      MOV     K22 D1902
      G.OUTPUT U5 D1900 D1911 M4010
2524  LD      M4010
      MPS
      ANI     M4011
      SET     M4110
      MPP
      AND     M4011
      SET     M4111
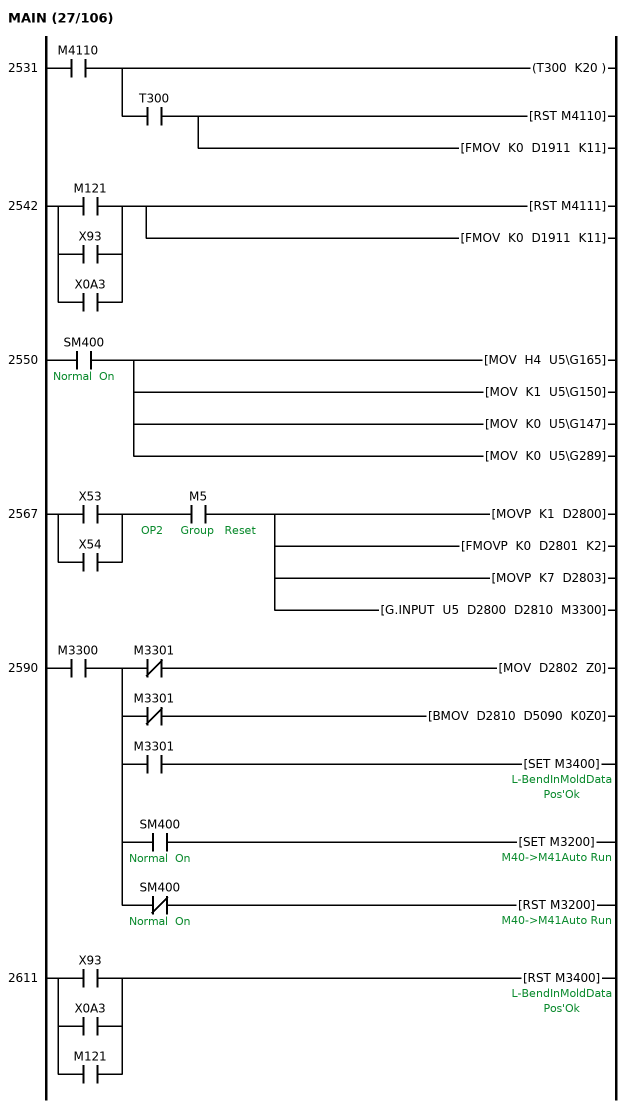
2531  LD      M4110
      OUT     T300 K20
      AND     T300
      RST     M4110
      FMOV    K0 D1911 K11
2542  LD      M121
      OR      X93
      OR      X0A3
      RST     M4111
      FMOV    K0 D1911 K11
2550  LD      SM400  ; Normal  On
      MOV     H4 U5\G165
      MOV     K1 U5\G150
      MOV     K0 U5\G147
      MOV     K0 U5\G289
2567  LD      X53
      OR      X54
      AND     M5  ; OP2     Group   Reset
      MOVP    K1 D2800
      FMOVP   K0 D2801 K2
      MOVP    K7 D2803
      G.INPUT U5 D2800 D2810 M3300
2590  LD      M3300
      MPS
      ANI     M3301
      MOV     D2802 Z0
      MRD
      ANI     M3301
      BMOV    D2810 D5090 K0Z0
      MRD
      AND     M3301
      SET     M3400  ; L-BendInMoldDataPos'Ok
      MRD
      AND     SM400  ; Normal  On
      SET     M3200  ; M40->M41Auto Run
      MPP
      ANI     SM400  ; Normal  On
      RST     M3200  ; M40->M41Auto Run
2611  LD      X93
      OR      X0A3
      OR      M121
      RST     M3400  ; L-BendInMoldDataPos'Ok
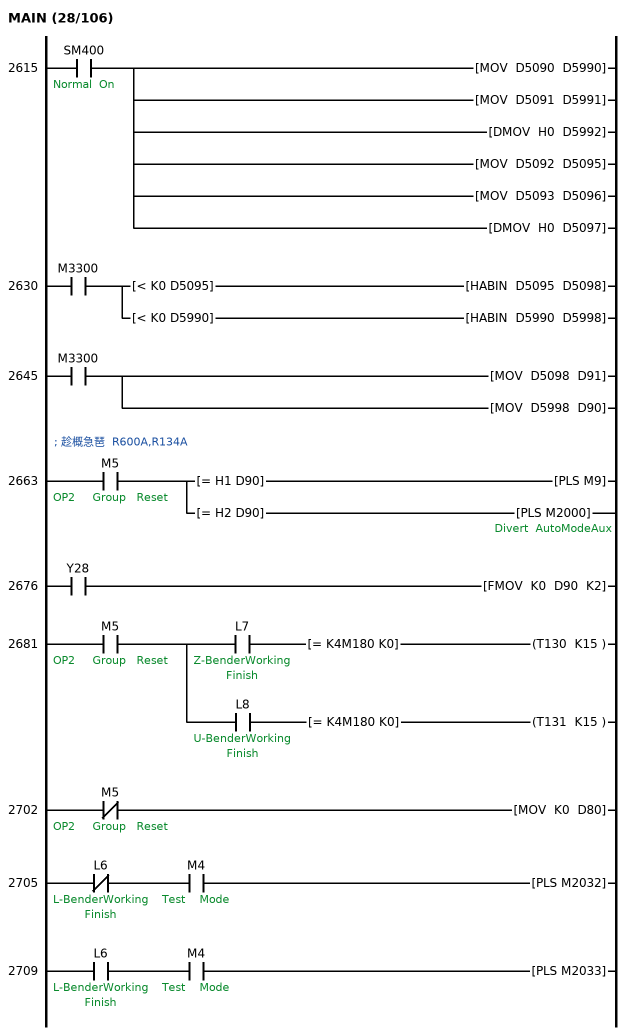
2615  LD      SM400  ; Normal  On
      MOV     D5090 D5990
      MOV     D5091 D5991
      DMOV    H0 D5992
      MOV     D5092 D5095
      MOV     D5093 D5096
      DMOV    H0 D5097
2630  LD      M3300
      MPS
      AND<    K0 D5095
      HABIN   D5095 D5098
      MPP
      AND<    K0 D5990
      HABIN   D5990 D5998
2645  LD      M3300
      MOV     D5098 D91
      MOV     D5998 D90
; 냉매선택  R600A,R134A
2663  LD      M5  ; OP2     Group   Reset
      MPS
      AND=    H1 D90
      PLS     M9
      MPP
      AND=    H2 D90
      PLS     M2000  ; Divert  AutoModeAux
2676  LD      Y28
      FMOV    K0 D90 K2
2681  LD      M5  ; OP2     Group   Reset
      MPS
      AND     L7  ; Z-BenderWorking Finish
      AND=    K4M180 K0
      OUT     T130 K15
      MPP
      AND     L8  ; U-BenderWorking Finish
      AND=    K4M180 K0
      OUT     T131 K15
2702  LDI     M5  ; OP2     Group   Reset
      MOV     K0 D80
2705  LDI     L6  ; L-BenderWorking Finish
      AND     M4  ; Test    Mode
      PLS     M2032
2709  LD      L6  ; L-BenderWorking Finish
      AND     M4  ; Test    Mode
      PLS     M2033
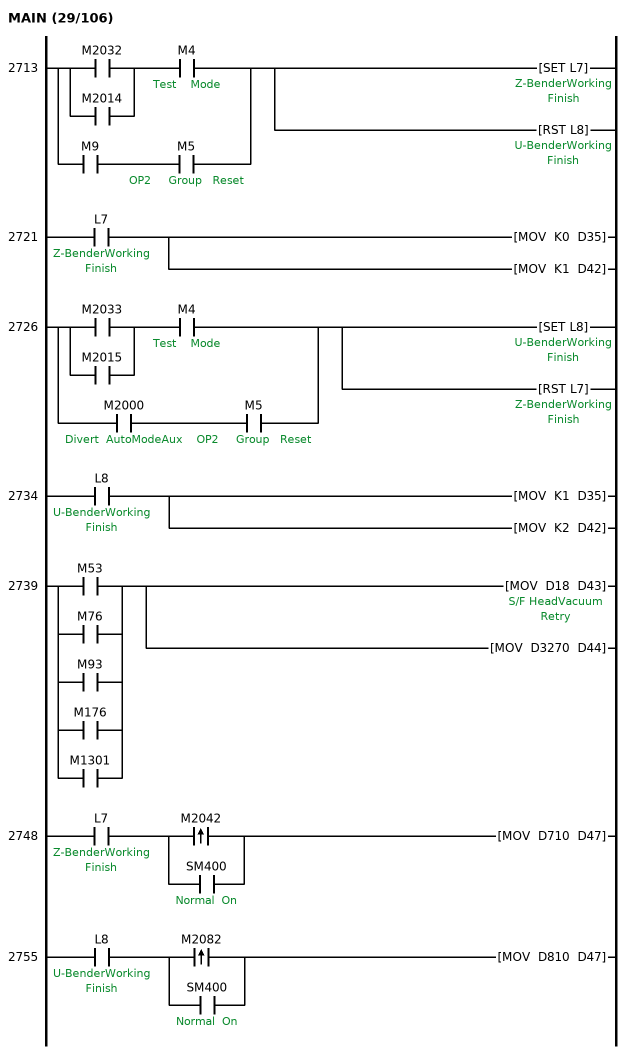
2713  LD      M2032
      OR      M2014
      AND     M4  ; Test    Mode
      LD      M9
      AND     M5  ; OP2     Group   Reset
      ORB
      SET     L7  ; Z-BenderWorking Finish
      RST     L8  ; U-BenderWorking Finish
2721  LD      L7  ; Z-BenderWorking Finish
      MOV     K0 D35
      MOV     K1 D42
2726  LD      M2033
      OR      M2015
      AND     M4  ; Test    Mode
      LD      M2000  ; Divert  AutoModeAux
      AND     M5  ; OP2     Group   Reset
      ORB
      SET     L8  ; U-BenderWorking Finish
      RST     L7  ; Z-BenderWorking Finish
2734  LD      L8  ; U-BenderWorking Finish
      MOV     K1 D35
      MOV     K2 D42
2739  LD      M53
      OR      M76
      OR      M93
      OR      M176
      OR      M1301
      MOV     D18 D43  ; S/F HeadVacuum  Retry
      MOV     D3270 D44
2748  LD      L7  ; Z-BenderWorking Finish
      LDP     M2042
      OR      SM400  ; Normal  On
      ANB
      MOV     D710 D47
2755  LD      L8  ; U-BenderWorking Finish
      LDP     M2082
      OR      SM400  ; Normal  On
      ANB
      MOV     D810 D47
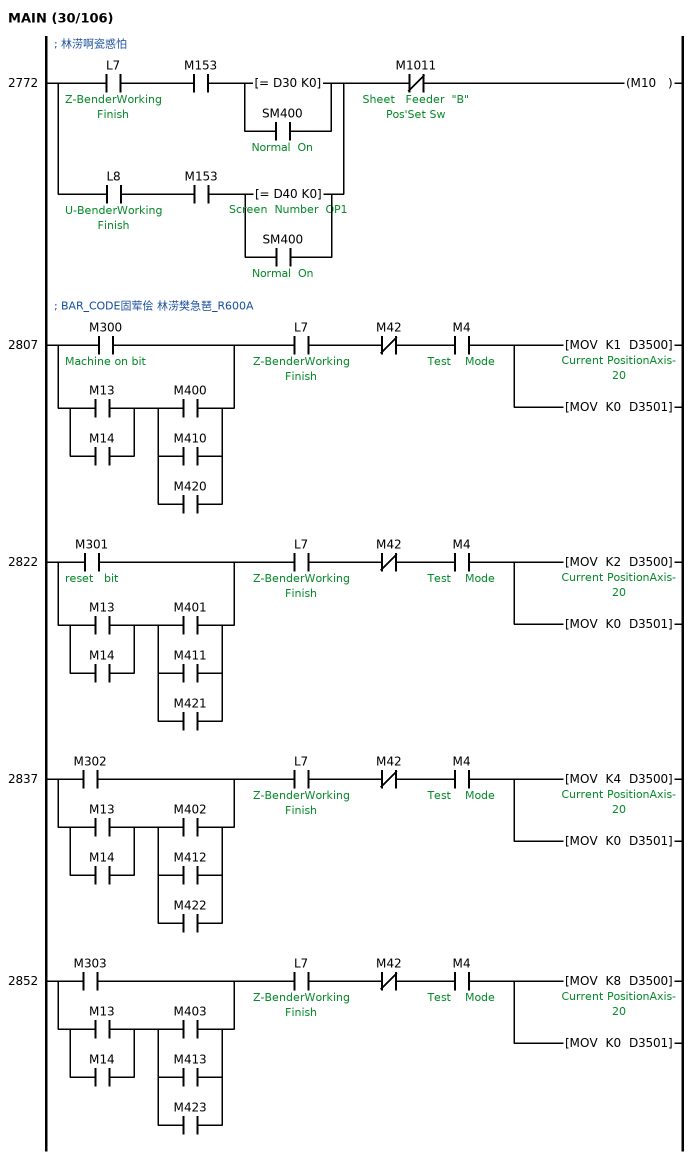
; 주입가능상태
; 
2772  LD      L7  ; Z-BenderWorking Finish
      AND     M153
      LD=     D30 K0
      OR      SM400  ; Normal  On
      ANB
      LD      L8  ; U-BenderWorking Finish
      AND     M153
      LD=     D40 K0  ; Screen  Number  OP1
      OR      SM400  ; Normal  On
      ANB
      ORB
      ANI     M1011  ; Sheet   Feeder  "B" Pos'Set Sw
      OUT     M10
; BAR_CODE미사용 주입량선택_R600A
2807  LD      M300  ; Machine on bit
      LD      M13
      OR      M14
      LD      M400
      OR      M410
      OR      M420
      ANB
      ORB
      AND     L7  ; Z-BenderWorking Finish
      ANI     M42
      AND     M4  ; Test    Mode
      MOV     K1 D3500  ; Current PositionAxis-20
      MOV     K0 D3501
2822  LD      M301  ; reset   bit
      LD      M13
      OR      M14
      LD      M401
      OR      M411
      OR      M421
      ANB
      ORB
      AND     L7  ; Z-BenderWorking Finish
      ANI     M42
      AND     M4  ; Test    Mode
      MOV     K2 D3500
      MOV     K0 D3501
2837  LD      M302
      LD      M13
      OR      M14
      LD      M402
      OR      M412
      OR      M422
      ANB
      ORB
      AND     L7  ; Z-BenderWorking Finish
      ANI     M42
      AND     M4  ; Test    Mode
      MOV     K4 D3500
      MOV     K0 D3501
2852  LD      M303
      LD      M13
      OR      M14
      LD      M403
      OR      M413
      OR      M423
      ANB
      ORB
      AND     L7  ; Z-BenderWorking Finish
      ANI     M42
      AND     M4  ; Test    Mode
      MOV     K8 D3500
      MOV     K0 D3501
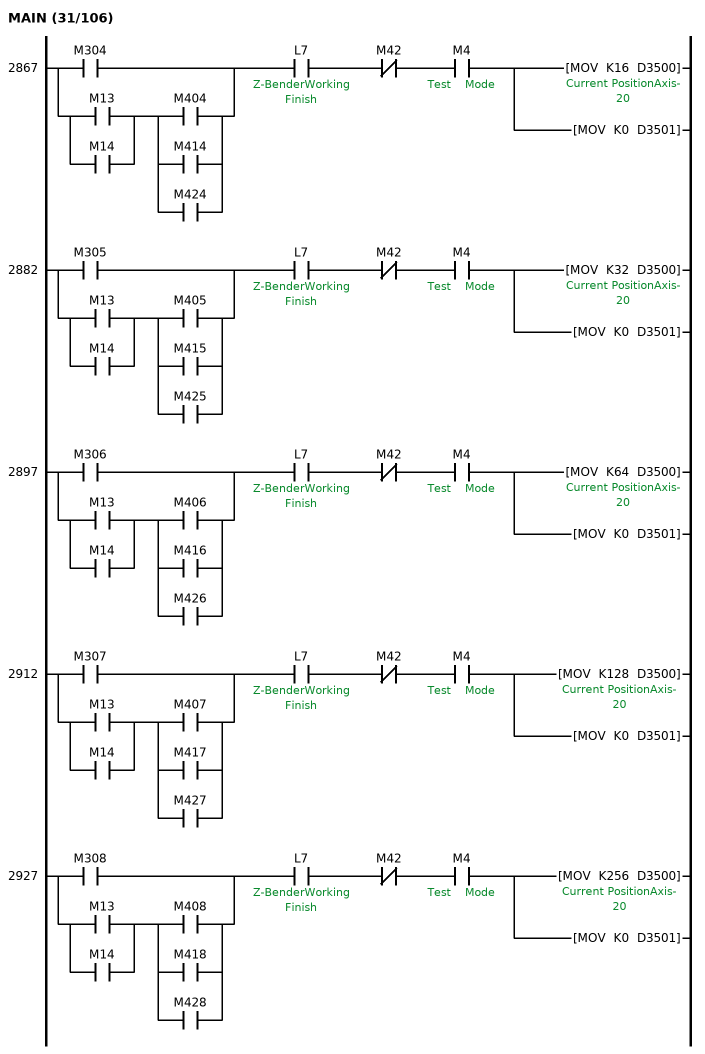
2867  LD      M304
      LD      M13
      OR      M14
      LD      M404
      OR      M414
      OR      M424
      ANB
      ORB
      AND     L7  ; Z-BenderWorking Finish
      ANI     M42
      AND     M4  ; Test    Mode
      MOV     K16 D3500
      MOV     K0 D3501
2882  LD      M305
      LD      M13
      OR      M14
      LD      M405
      OR      M415
      OR      M425
      ANB
      ORB
      AND     L7  ; Z-BenderWorking Finish
      ANI     M42
      AND     M4  ; Test    Mode
      MOV     K32 D3500
      MOV     K0 D3501
2897  LD      M306
      LD      M13
      OR      M14
      LD      M406
      OR      M416
      OR      M426
      ANB
      ORB
      AND     L7  ; Z-BenderWorking Finish
      ANI     M42
      AND     M4  ; Test    Mode
      MOV     K64 D3500
      MOV     K0 D3501
2912  LD      M307
      LD      M13
      OR      M14
      LD      M407
      OR      M417
      OR      M427
      ANB
      ORB
      AND     L7  ; Z-BenderWorking Finish
      ANI     M42
      AND     M4  ; Test    Mode
      MOV     K128 D3500
      MOV     K0 D3501
2927  LD      M308
      LD      M13
      OR      M14
      LD      M408
      OR      M418
      OR      M428
      ANB
      ORB
      AND     L7  ; Z-BenderWorking Finish
      ANI     M42
      AND     M4  ; Test    Mode
      MOV     K256 D3500
      MOV     K0 D3501
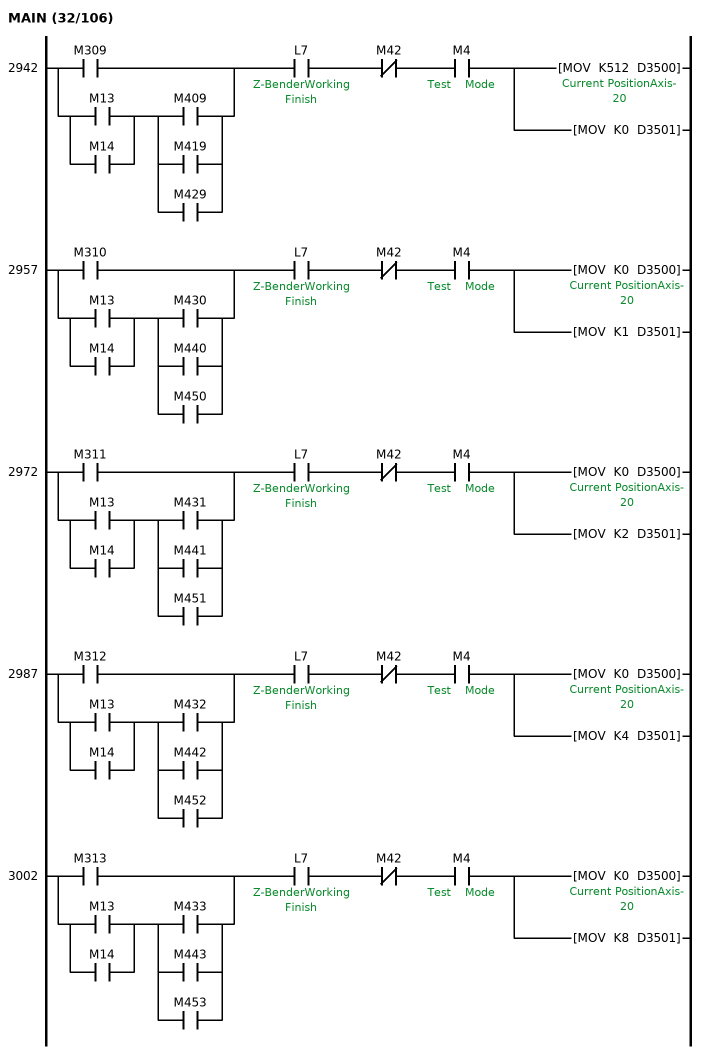
2942  LD      M309
      LD      M13
      OR      M14
      LD      M409
      OR      M419
      OR      M429
      ANB
      ORB
      AND     L7  ; Z-BenderWorking Finish
      ANI     M42
      AND     M4  ; Test    Mode
      MOV     K512 D3500
      MOV     K0 D3501
2957  LD      M310
      LD      M13
      OR      M14
      LD      M430
      OR      M440
      OR      M450
      ANB
      ORB
      AND     L7  ; Z-BenderWorking Finish
      ANI     M42
      AND     M4  ; Test    Mode
      MOV     K0 D3500
      MOV     K1 D3501
2972  LD      M311
      LD      M13
      OR      M14
      LD      M431
      OR      M441
      OR      M451
      ANB
      ORB
      AND     L7  ; Z-BenderWorking Finish
      ANI     M42
      AND     M4  ; Test    Mode
      MOV     K0 D3500
      MOV     K2 D3501
2987  LD      M312
      LD      M13
      OR      M14
      LD      M432
      OR      M442
      OR      M452
      ANB
      ORB
      AND     L7  ; Z-BenderWorking Finish
      ANI     M42
      AND     M4  ; Test    Mode
      MOV     K0 D3500
      MOV     K4 D3501
3002  LD      M313
      LD      M13
      OR      M14
      LD      M433
      OR      M443
      OR      M453
      ANB
      ORB
      AND     L7  ; Z-BenderWorking Finish
      ANI     M42
      AND     M4  ; Test    Mode
      MOV     K0 D3500
      MOV     K8 D3501
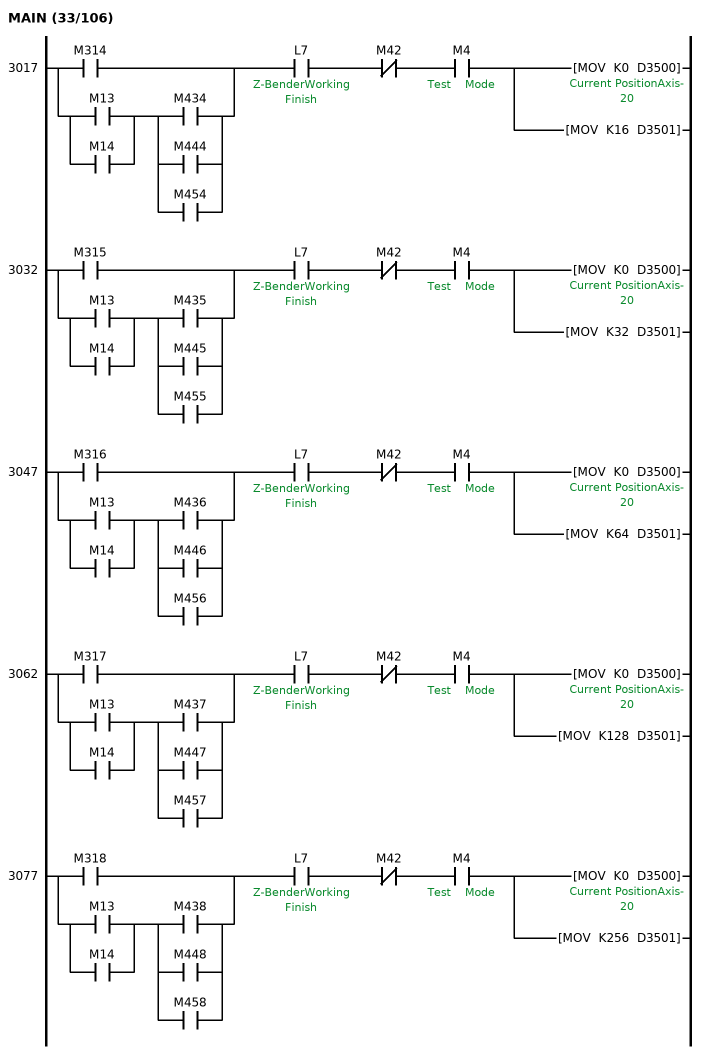
3017  LD      M314
      LD      M13
      OR      M14
      LD      M434
      OR      M444
      OR      M454
      ANB
      ORB
      AND     L7  ; Z-BenderWorking Finish
      ANI     M42
      AND     M4  ; Test    Mode
      MOV     K0 D3500
      MOV     K16 D3501
3032  LD      M315
      LD      M13
      OR      M14
      LD      M435
      OR      M445
      OR      M455
      ANB
      ORB
      AND     L7  ; Z-BenderWorking Finish
      ANI     M42
      AND     M4  ; Test    Mode
      MOV     K0 D3500
      MOV     K32 D3501
3047  LD      M316
      LD      M13
      OR      M14
      LD      M436
      OR      M446
      OR      M456
      ANB
      ORB
      AND     L7  ; Z-BenderWorking Finish
      ANI     M42
      AND     M4  ; Test    Mode
      MOV     K0 D3500
      MOV     K64 D3501
3062  LD      M317
      LD      M13
      OR      M14
      LD      M437
      OR      M447
      OR      M457
      ANB
      ORB
      AND     L7  ; Z-BenderWorking Finish
      ANI     M42
      AND     M4  ; Test    Mode
      MOV     K0 D3500
      MOV     K128 D3501
3077  LD      M318
      LD      M13
      OR      M14
      LD      M438
      OR      M448
      OR      M458
      ANB
      ORB
      AND     L7  ; Z-BenderWorking Finish
      ANI     M42
      AND     M4  ; Test    Mode
      MOV     K0 D3500
      MOV     K256 D3501
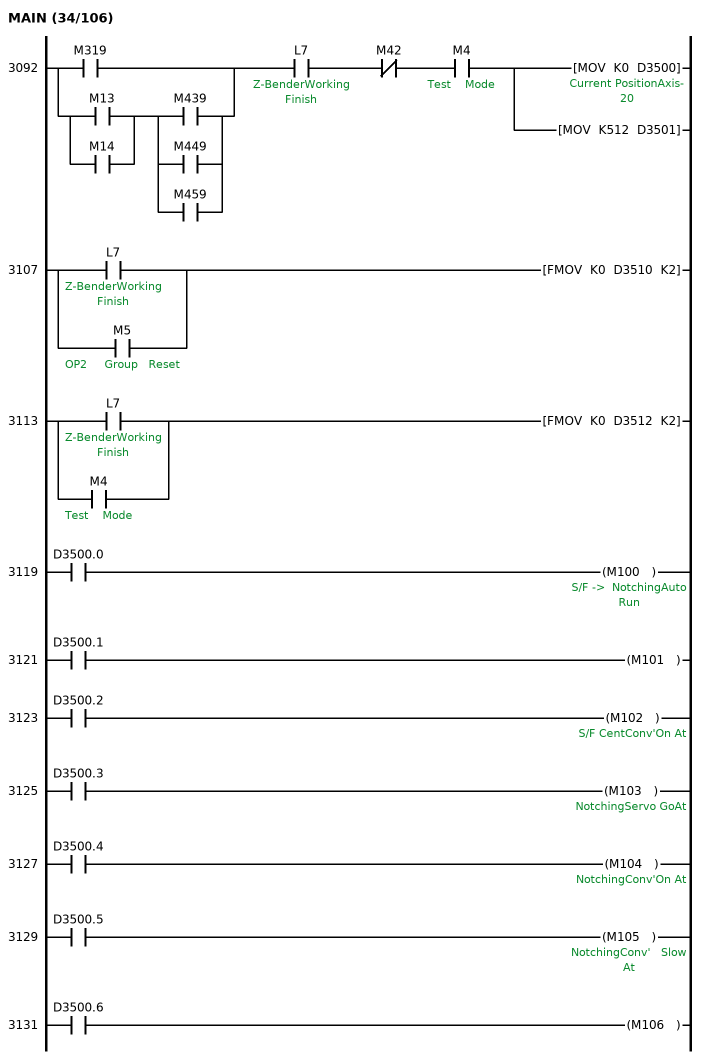
3092  LD      M319
      LD      M13
      OR      M14
      LD      M439
      OR      M449
      OR      M459
      ANB
      ORB
      AND     L7  ; Z-BenderWorking Finish
      ANI     M42
      AND     M4  ; Test    Mode
      MOV     K0 D3500
      MOV     K512 D3501
3107  LD      L7  ; Z-BenderWorking Finish
      OR      M5  ; OP2     Group   Reset
      FMOV    K0 D3510 K2
3113  LD      L7  ; Z-BenderWorking Finish
      OR      M4  ; Test    Mode
      FMOV    K0 D3512 K2
3119  LD      D3500.0
      OUT     M100  ; S/F ->  NotchingAuto Run
3121  LD      D3500.1
      OUT     M101
3123  LD      D3500.2
      OUT     M102  ; S/F CentConv'On At
3125  LD      D3500.3
      OUT     M103  ; NotchingServo GoAt
3127  LD      D3500.4
      OUT     M104  ; NotchingConv'On At
3129  LD      D3500.5
      OUT     M105  ; NotchingConv'   Slow At
3131  LD      D3500.6
      OUT     M106
